{attribute 'linkalways'} 
{attribute 'no_explicit_call' := 'This FB is a CLASS and must be accessed using methods or properties'}
{attribute 'enable_dynamic_creation'}
FUNCTION_BLOCK FINAL FLOOR_LREAL EXTENDS Node
VAR
	in : _LREAL(0.0);
	out : _LREAL(0.0);
END_VAR

METHOD PUBLIC Clone : I_Node
VAR
	pNode : POINTER TO FLOOR_LREAL;
END_VAR
pNode := __NEW(FLOOR_LREAL);
Clone := pNode^;
END_METHOD

METHOD FB_init : BOOL
VAR_INPUT
	bInitRetains : BOOL; // if TRUE, the retain variables are initialized (warm start / cold start)
	bInCopyCode : BOOL;  // if TRUE, the instance afterwards gets moved into the copy code (online change)
END_VAR
AddInput('in',THIS^.in);
AddOutput('out', THIS^.out);
END_METHOD

METHOD PROTECTED OnExecute
VAR
END_VAR
out.Value := FLOOR(in.Value);
END_METHOD

END_FUNCTION_BLOCK

(* stored: Version 1.1.0.1, ProductVersion 3.1.4024.15
   POU FLOOR_LREAL: Id {c545af4b-dce3-4874-98c6-fab206815808}, SpecialFunc None
   Folder Constructor: Id {f2ca7103-c6a5-4c21-9abf-ff1f8e73d60e}
   Method Clone: Id {2c1ad381-05d2-4237-9df8-be935543f71d}
   Method FB_init: Id {db79a9d5-0625-4391-b436-17ade98a4492}
   Method OnExecute: Id {a9aa84ec-6958-4fd0-a378-fca28ff0281a} *)
